Staubli VAL3: GenericConv.pjx

--- GenericConv.pjx ---
Parameters version=s7.6 stackSize=5000 millimeterUnit=true
Program file=checkTrackArea.pgx
Program file=conveyor.pgx
Program file=create.pgx
Program file=disableQueue.pgx
Program file=enableQueue.pgx
Program file=fillQueue.pgx
Program file=flushQueue.pgx
Program file=getConvFrame.pgx
Program file=getDetectDist.pgx
Program file=getDetectFrame.pgx
Program file=getDistance.pgx
Program file=getErrorMessage.pgx
Program file=getNextID.pgx
Program file=getObjectData.pgx
Program file=getObjectLatch.pgx
Program file=getObjectOffset.pgx
Program file=getObjectPos.pgx
Program file=getStatus.pgx
Program file=getTravelDist.pgx
Program file=init.pgx
Program file=kill.pgx
Program file=releaseObject.pgx
Program file=removePart.pgx
Program file=reset.pgx
Program file=setCalibrating.pgx
Program file=setConveyor.pgx
Program file=setObjectInUse.pgx
Program file=start.pgx
Program file=stop.pgx
Program file=teach.pgx
Program file=whichObjectUsed.pgx
Data file=GenericConv.dtx
Library alias=cfg path=Disk://Tracking/config/config.pjx
Library alias=det path=Disk://Tracking/Templates/GenericDetect/GenericDetect.pjx autoload=false
Library alias=enc path=Disk://Tracking/Templates/GenericEnc/GenericEnc.pjx autoload=false
Library alias=geometry path=Disk://Tracking/Templates/Geometry/Geometry.pjx autoload=false
Library alias=swap path=Disk://Tracking/Swap/Swap.pjx
Library alias=ut path=Disk://Tracking/Tools/util/util.pjx
Library alias=lang path=Disk://Tracking/language/english/english.pjx
Library alias=out path=Disk://Tracking/io/outputs/outputs.pjx

--- kill.pgx ---
public program kill(num x_nConvNum)
begin
  call enc:kill()
  taskKill(sTASK[0]+toString("",x_nConvNum))
  call det:kill()
end

--- releaseObject.pgx ---
public program releaseObject(num x_nIdx)
  local string l_str
  local num l_nQueue
  local string l_sMessage
begin
  // This programs is used to count how many users have accessed
  // to the data of an object in the queue
  //
  // Input param
  //  x_nIdx       : Index of the object in the queue
  //
  // Output param
  //  none
  //
  //----------------------------------------------------------------
  //
  nNumbOfUser[x_nIdx]=max(0,nNumbOfUser[x_nIdx]-1)
  if (roundDown(nNumbOfUser[x_nIdx])<=0)
    nQueueID[x_nIdx]=-1
    //
    if bAnd(cfg:nLog,cfg:nLOGQUEUE)==cfg:nLOGQUEUE and bLOG
      ? sConvNum+"(releaseObject)>>"
      ? "           -------------------------Remove Part------------------------"
      ? "           |Index|  ID | latch value |     x    |     y    |    rz    |"
      ? "           ------------------------------------------------------------"
      for l_nQueue=0 to nBufferSize-1
        if nQueueID[l_nQueue]>=0
          l_sMessage="           | "+toString("3.0",l_nQueue)+" | "+toString("3.0",nQueueID[l_nQueue])+" | "+toString("11.2",nEncLatchedVal[l_nQueue])+" | "
          l_sMessage=l_sMessage+toString("8.2",trDetectedCoord[l_nQueue].x)+" | "+toString("8.2",trDetectedCoord[l_nQueue].y)+" | "+toString("8.2",trDetectedCoord[l_nQueue].rz)+" |"
          ? l_sMessage
        endIf
      endFor
      ? "           ------------------------------------------------------------"
      ? ""
    endIf
    //
  endIf
  if bAnd(cfg:nLog,cfg:nLOGMOTION)==cfg:nLOGMOTION
    l_str=sConvNum+"(releaseObject)>>Request to release object @ position "+toString("",x_nIdx)+" in queue, nbUser="
    l_str=l_str+toString("",nNumbOfUser[x_nIdx])
    ? l_str
  endIf
end
